{attribute addProperty BoxType "EL6002-0000-0016"}
{attribute addProperty Id "CtrlAT %Q*Ctrl_9717E367445.51Data_OutAT %Q*ARRAY[0 ..21] OF USINT176220"}
{attribute addProperty CRC "2316584694"}
{attribute addProperty SizeInBites "220"}
{attribute addProperty SizeInBytes "27.5"}
TYPE COM_Outputs_Channel_60FF225E :
STRUCT
	{attribute addProperty Name "Ctrl"}
	Ctrl AT %Q* : Ctrl_9717E367;
	{attribute addProperty Name "Data_Out"}
	Data_Out AT %Q* : ARRAY[0 ..21] OF USINT;
END_STRUCT
END_TYPE

(* stored: Version 1.2.0.0, ProductVersion 3.1.4024.9
   DUT COM_Outputs_Channel_60FF225E: Id {fca7bcf5-10c6-4904-8634-efd54690520e} *)
